{attribute 'enable_dynamic_creation'}
FUNCTION_BLOCK FB_WaitForConditionCommand IMPLEMENTS I_Command
VAR
	condition : I_BoolValue;
	minWaitTime : TIME;
	maxWaitTime : TIME;
	minWaiter : TON;
	maxWaiter : TON;
	_Description : STRING;
END_VAR

{attribute 'monitoring' := 'call'}
PROPERTY Description : STRING
GET
Description := _Description;
END_GET
END_PROPERTY

METHOD Execute : E_ProgressStatus
minWaiter(IN := TRUE, PT := minWaitTime);
maxWaiter(IN := maxWaitTime > T#0S, PT := maxWaitTime);

IF ((condition.Value AND minWaiter.Q) OR maxWaiter.Q) THEN
	Execute := E_ProgressStatus.Completed;
ELSE
	Execute := E_ProgressStatus.Running;
END_IF
END_METHOD

//FB_Init is always available implicitly and it is used primarily for initialization.
//The return value is not evaluated. For a specific influence, you can also declare the
//methods explicitly and provide additional code there with the standard initialization
//code. You can evaluate the return value.
METHOD FB_Init: BOOL
VAR_INPUT
    bInitRetains: BOOL; // TRUE: the retain variables are initialized (reset warm / reset cold)
    bInCopyCode: BOOL;  // TRUE: the instance will be copied to the copy code afterward (online change)   
	
	condition : I_BoolValue;
	minWaitTime : TIME;
	maxWaitTime : TIME;
	description : STRING;
END_VAR
THIS^.condition := condition;
THIS^.minWaitTime := minWaitTime;
THIS^.maxWaitTime := maxWaitTime;
_Description := description;
END_METHOD

METHOD Reset
VAR_INPUT
END_VAR
minWaiter(IN := FALSE);
maxWaiter(IN := FALSE);
END_METHOD

END_FUNCTION_BLOCK

(* stored: Version 1.1.0.1
   POU FB_WaitForConditionCommand: Id {1a081878-4346-4de3-9264-4856341ae2ac}, SpecialFunc None
   Property Description: Id {ead1b661-5d60-49be-89d6-b3a5c12d38e2}
   Get Get: Id {096b513b-77e8-44cc-b4e3-427cadc56271}
   Method Execute: Id {e374f8e9-fa4a-47b1-84a5-cd13345a671e}
   Method FB_Init: Id {5442f766-a903-4c70-9f98-111841e7482a}
   Method Reset: Id {f626ef0a-73ce-4bb4-8759-051c6de8a162} *)
